FUNCTION F_deg2rad : LREAL
VAR_INPUT
	fInputRad : LREAL;
END_VAR
VAR
	pi : LREAL := 3.14159265;
END_VAR

F_deg2rad := (pi/180)*fInputRad;

END_FUNCTION

(* stored: Version 1.1.0.1, ProductVersion 3.1.4024.12
   POU F_deg2rad: Id {f03115d6-0cc3-427c-baf0-660c1dc69a12}, SpecialFunc None *)
